{attribute 'strict'}
{attribute 'to_string'}
TYPE E_VisuCtrlAxisImgType :
(
	AXIS_TYPE_BECKHOFF_SERVO_AM30XX 	:= 0,	(*  *)
	AXIS_TYPE_BECKHOFF_SERVO_AM80XX 	:= 10,	(*  *)
	AXIS_TYPE_BECKHOFF_SERVO_AM81XX 	:= 20,	(*  *)
	AXIS_TYPE_BECKHOFF_SERVO_AM85XX		:= 30,	(*  *)
	AXIS_TYPE_BECKHOFF_SERVO_AM87XX		:= 40,	(*  *)
	AXIS_TYPE_BECKHOFF_SERVO_AM88XX		:= 50,	(*  *)
	AXIS_TYPE_BECKHOFF_SERVO_AMI812X	:= 60,	(*  *)
	AXIS_TYPE_BECKHOFF_SERVO_AMP80XX	:= 70,	(*  *)
	AXIS_TYPE_BECKHOFF_STEPPER_AG1000 	:= 80,	(*  *)
	AXIS_TYPE_BECKHOFF_STEPPER_AG2250 	:= 90,	(*  *)
	AXIS_TYPE_BECKHOFF_STEPPER_ASXXX 	:= 100,	(*  *)
	AXIS_TYPE_FAULHABER_LM_1257			:= 110,	(*  *)
	AXIS_TYPE_JENNY_SCIENCE_ELAX		:= 120,	(*  *)
	AXIS_TYPE_JENNY_SCIENCE_LINAX_LXC	:= 130,	(*  *)
	AXIS_TYPE_JENNY_SCIENCE_LINAX_LXS	:= 140,	(*  *)
	AXIS_TYPE_JENNY_SCIENCE_LINAX_LXU	:= 150,	(*  *)
	AXIS_TYPE_JENNY_SCIENCE_LINAX_LXE	:= 160,	(*  *)
	AXIS_TYPE_JENNY_SCIENCE_ROTAX_28	:= 170,	(*  *)
	AXIS_TYPE_JENNY_SCIENCE_ROTAX_50	:= 180,	(*  *)
	AXIS_TYPE_JENNY_SCIENCE_ROTAX_110	:= 190,	(*  *)
	AXIS_TYPE_BECKHOFF_XTS_MOVER		:= 200	(*  *)
);
END_TYPE

(* stored: Version 1.1.0.1, ProductVersion 3.1.4024.12
   DUT E_VisuCtrlAxisImgType: Id {a0fad3e0-c26a-4236-bc29-216e46de8c1c} *)
